// TIA Portal project "P8" (V17)

(* hardware
DEVICE "S7-1500/ET200MP station_1"  S7-1500 station
   slot 0: "Rail_0"  Rack  6ES7 590-1***0-0AA0
   slot 1: "PLC_1"  CPU 1512C-1 PN  6ES7 512-1CK01-0AB0  V2.9
      slot 3: "CPU display_1"  6ES7591-1AA00-0AA0
      slot 32768: "PROFINET interface_1"  X1
         slot 32769: "Port_1"  X1 P1
         slot 32770: "Port_2"  X1 P2
      slot 34817: "Virtual CP interface port_1"  Virtual CP interface port  Virtual CP interface port
*)

// ===== PLC "PLC_1"  CPU 1512C-1 PN =====

VAR_GLOBAL   // PLC tag table "Default tag table"
   "Enable Command Scaling" AT %M0.0 : Bool;
   "Bipolar Selection-Scaling" AT %M0.1 : Bool;
   "Bipolar Selection-Unscaling" AT %M0.2 : Bool;
   "Actual Valvule from for sensor" AT %MW10 : Int;
   "Error word-Scaling" AT %MW12 : Word;
   "Scaled output" AT %MD20 : Real;
   "Enable command Unscaling" AT %M1.0 : Bool;
   "Given value from the display" AT %MD24 : Real;
   "Error word-Unscaling" AT %MW16 : Word;
   "Unscaled output" AT %MW26 : Int;
END_VAR

ORGANIZATION_BLOCK "Main"   // OB1, LAD, ProgramCycle
TITLE = "Main Program Sweep (Cycle)"
{ S7_Optimized_Access := 'TRUE' }
VERSION : 0.1
   VAR_INPUT
      Initial_Call : Bool;   // Initial call of this OB
      Remanence : Bool;   // =True, if remanent data are available
   END_VAR
BEGIN

REGION Network 1
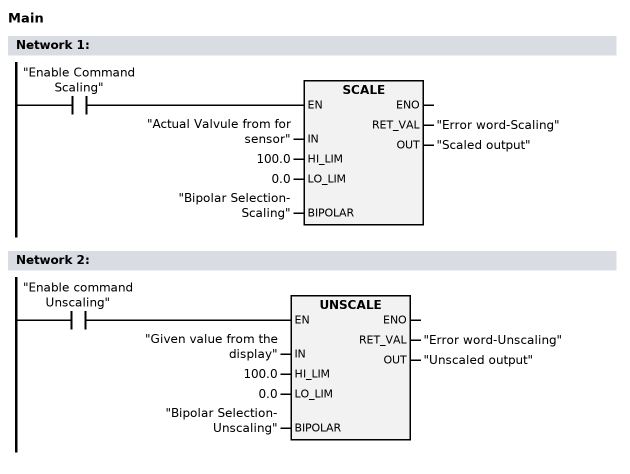
   IF "Enable Command Scaling" THEN
       "Error word-Scaling" := SCALE(IN := "Actual Valvule from for sensor",
                               HI_LIM := 100.0,
                               LO_LIM := 0.0,
                               BIPOLAR := "Bipolar Selection-Scaling",
                               OUT => "Scaled output");
   END_IF;
END_REGION

REGION Network 2
   IF "Enable command Unscaling" THEN
       "Error word-Unscaling" := UNSCALE(IN := "Given value from the display",
                               HI_LIM := 100.0,
                               LO_LIM := 0.0,
                               BIPOLAR := "Bipolar Selection-Unscaling",
                               OUT => "Unscaled output");
   END_IF;
END_REGION
END_ORGANIZATION_BLOCK